FUNCTION ACOSD : LREAL
VAR_INPUT
	COSVAL:LREAL;
END_VAR
VAR
END_VAR

ACOSD:=RAD_TO_DEG(ACOS(COSVAL));

END_FUNCTION

(* stored: Version 1.1.0.1, ProductVersion 3.1.4024.12
   POU ACOSD: Id {cec39ffe-144d-4802-9afb-98ee0757f3ff}, SpecialFunc None *)
